// TIA Portal V17 export
// export: Created 2025-03-12T15:37:05.3598462Z, ExportSetting WithDefaults, DisplayName Totally Integrated Automation Portal, DisplayVersion V17 Update 8, DisplayName TIA Portal Openness, DisplayVersion V17 Update 8, DisplayName TIA Portal Version Control Interface, DisplayVersion V17, DisplayName SINAMICS Startdrive Advanced, DisplayVersion V17 SP2, DisplayName SINAMICS Startdrive G110M, G120, G120C, G120D, G120P, G115D, DisplayVersion V17 SP2, DisplayName SINAMICS Startdrive G130, G150, S120, S150, SINAMICS MV, S210, DisplayVersion V17 SP2, DisplayName STEP 7 Professional, DisplayVersion V17 Update 8, DisplayName SINUMERIK ONE STEP 7 Toolbox, DisplayVersion V17 Update 12, DisplayName SINUMERIK 840D sl STEP 7 Toolbox, DisplayVersion V17 Update 12, DisplayName STEP 7 Safety, DisplayVersion V17 Update 6, DisplayName WinCC Advanced, DisplayVersion V17 Update 8
TYPE "READ_CNC_MEMORY_1"
// stored: IsFailsafeCompliant false
   STRUCT
      Read : Bool;   // Lesen der Daten angefordert
      Busy : Bool;   // Aufruf SFC51 ist aktiv
      ListenId : Word;   // Listen-ID, die ausgelesen werden soll, alle Speicherbereiche (1, 3)
      ListenIndex : Word;   // Index fuer den Datensatz, hier Anwenderspeicher
      RetVal : Int;   // Returnwert fuerdas Auslesen des Anwender-Spechers
      SZL_HEADER : Struct
         LengthDataBlock : Word;   // Laenge eines Datensatzes
         CountDataBlock : Word;   // Anzahl vorhandener / gelesener Datensaetze
      END_STRUCT;
   END_STRUCT;
END_TYPE
